// TIA Portal project "GirelloFB" (V16)

(* hardware
DEVICE "S7-1200 station_1"  S7-1200 Station
   slot 0: "Telaio di montaggio_0"  S7-1200 Rack  Rack  V1.0
   slot 1: "PLC_1"  CPU 1214C DC/DC/Rly  6ES7 214-1HG40-0XB0  V4.1
*)

// ===== PLC "PLC_1"  CPU 1214C DC/DC/Rly =====

VAR_GLOBAL   // PLC tag table "Tabella delle variabili standard"
   "START_1" AT %I0.0 : Bool;
   "S1_1" AT %I0.1 : Bool;
   "S2_1" AT %I0.2 : Bool;
   "S3_1" AT %I0.3 : Bool;
   "M_left_1" AT %Q0.0 : Bool;
   "M_right_1" AT %Q0.1 : Bool;
   "START_2" AT %I0.4 : Bool;
   "S1_2" AT %I0.5 : Bool;
   "S2_2" AT %I0.6 : Bool;
   "M_left_2" AT %Q0.2 : Bool;
   "M_right_2" AT %Q0.3 : Bool;
   "S3_2" AT %I0.7 : Bool;
END_VAR

VAR_GLOBAL CONSTANT   // PLC tag table "Tabella delle variabili standard"
   "TEMPO_TRASCORSO_T1_Girello1" : Time := T#3s;
   "TEMPO_TRASCORSO_T2_Girello1" : Time := T#8s;
   "TEMPO_TRASCORSO_T1_Girello2" : Time := T#5s;
   "TEMPO_TRASCORSO_T2_Girello2" : Time := T#10s;
END_VAR

DATA_BLOCK "Girello_DB_1"   // DB1
{ S7_Optimized_Access := 'TRUE' }
VERSION : 0.1
// stored: InstanceOfName Girello
"Girello"
BEGIN
END_DATA_BLOCK

DATA_BLOCK "Girello_DB_2"   // DB2
{ S7_Optimized_Access := 'TRUE' }
VERSION : 0.1
// stored: InstanceOfName Girello
"Girello"
BEGIN
END_DATA_BLOCK

FUNCTION_BLOCK "Girello"   // FB1, LAD
{ S7_Optimized_Access := 'TRUE' }
VERSION : 0.1
   VAR_INPUT
      START : Bool;
      S1 : Bool;
      S2 : Bool;
      S3 : Bool;
      TEMPO_TRASCORSO_T1 : Time;
      TEMPO_TRASCORSO_T2 : Time;
   END_VAR
   VAR_OUTPUT
      M_left : Bool;
      M_right : Bool;
   END_VAR
   VAR RETAIN
      HOME : Bool := true;
      ROTATE_TO_LEFT : Bool;
      POSITION_S2 : Bool;
      POSITION_S3 : Bool;
      ROTATE_TO_RIGHT : Bool;
   END_VAR
   VAR
      IEC_Timer_0_Instance_1 : TON_TIME;
      IEC_Timer_0_Instance_2 : TON_TIME;
   END_VAR
BEGIN

REGION Network 1
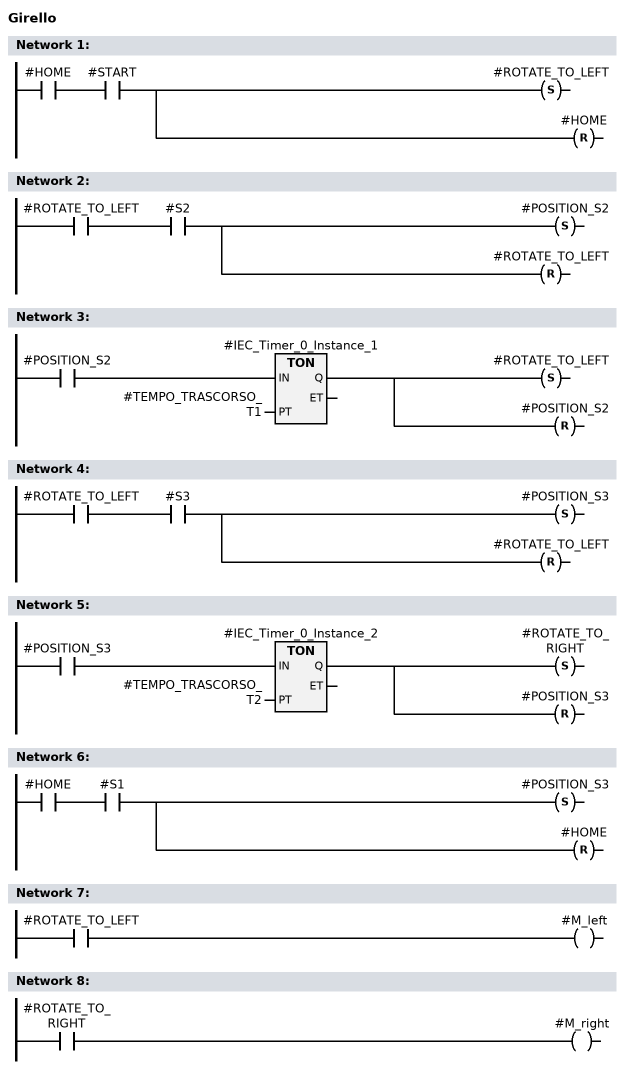
   RUNG wire#powerrail
      Contact( #HOME )
      Contact( #START )
      wire#w1
      S_Coil( #ROTATE_TO_LEFT )
   END_RUNG
   RUNG wire#w1
      R_Coil( #HOME )
   END_RUNG
   // the same network as SCL:
   IF #HOME AND #START THEN
       #ROTATE_TO_LEFT := TRUE;
       #HOME := FALSE;
   END_IF;
END_REGION

REGION Network 2
   RUNG wire#powerrail
      Contact( #ROTATE_TO_LEFT )
      Contact( #S2 )
      wire#w1
      S_Coil( #POSITION_S2 )
   END_RUNG
   RUNG wire#w1
      R_Coil( #ROTATE_TO_LEFT )
   END_RUNG
   // the same network as SCL:
   IF #ROTATE_TO_LEFT AND #S2 THEN
       #POSITION_S2 := TRUE;
       #ROTATE_TO_LEFT := FALSE;
   END_IF;
END_REGION

REGION Network 3
   #IEC_Timer_0_Instance_1(IN := #POSITION_S2, PT := #TEMPO_TRASCORSO_T1);   // TON
   IF #IEC_Timer_0_Instance_1.Q THEN
       #ROTATE_TO_LEFT := TRUE;
       #POSITION_S2 := FALSE;
   END_IF;
END_REGION

REGION Network 4
   RUNG wire#powerrail
      Contact( #ROTATE_TO_LEFT )
      Contact( #S3 )
      wire#w1
      S_Coil( #POSITION_S3 )
   END_RUNG
   RUNG wire#w1
      R_Coil( #ROTATE_TO_LEFT )
   END_RUNG
   // the same network as SCL:
   IF #ROTATE_TO_LEFT AND #S3 THEN
       #POSITION_S3 := TRUE;
       #ROTATE_TO_LEFT := FALSE;
   END_IF;
END_REGION

REGION Network 5
   #IEC_Timer_0_Instance_2(IN := #POSITION_S3, PT := #TEMPO_TRASCORSO_T2);   // TON
   IF #IEC_Timer_0_Instance_2.Q THEN
       #ROTATE_TO_RIGHT := TRUE;
       #POSITION_S3 := FALSE;
   END_IF;
END_REGION

REGION Network 6
   RUNG wire#powerrail
      Contact( #HOME )
      Contact( #S1 )
      wire#w1
      S_Coil( #POSITION_S3 )
   END_RUNG
   RUNG wire#w1
      R_Coil( #HOME )
   END_RUNG
   // the same network as SCL:
   IF #HOME AND #S1 THEN
       #POSITION_S3 := TRUE;
       #HOME := FALSE;
   END_IF;
END_REGION

REGION Network 7
   RUNG wire#powerrail
      Contact( #ROTATE_TO_LEFT )
      Coil( #M_left )
   END_RUNG
   // the same network as SCL:
   #M_left := #ROTATE_TO_LEFT;
END_REGION

REGION Network 8
   RUNG wire#powerrail
      Contact( #ROTATE_TO_RIGHT )
      Coil( #M_right )
   END_RUNG
   // the same network as SCL:
   #M_right := #ROTATE_TO_RIGHT;
END_REGION
END_FUNCTION_BLOCK

ORGANIZATION_BLOCK "Main"   // OB1, LAD, ProgramCycle
TITLE = "Main Program Sweep (Cycle)"
{ S7_Optimized_Access := 'TRUE' }
VERSION : 0.1
   VAR_INPUT
      Initial_Call : Bool;   // Initial call of this OB
      Remanence : Bool;   // =True, if remanent data are available
   END_VAR
BEGIN
END_ORGANIZATION_BLOCK

ORGANIZATION_BLOCK "Cyclic_Interrupt_50ms"   // OB30, LAD, CyclicInterrupt
{ S7_Optimized_Access := 'TRUE' }
VERSION : 0.1
   VAR_INPUT
      Initial_Call : Bool;   // Initial call of this OB
      Event_Count : Int;   // Events discarded
   END_VAR
BEGIN

REGION Network 1
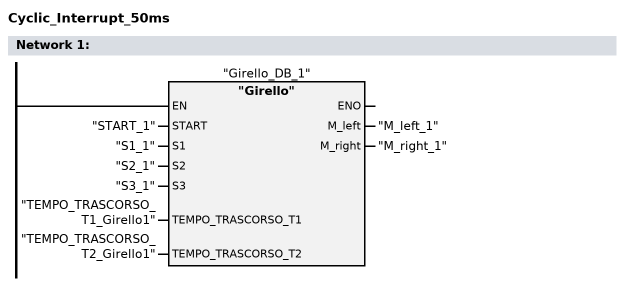
   RUNG wire#powerrail
      "Girello_DB_1"(START := "START_1", S1 := "S1_1", S2 := "S2_1", S3 := "S3_1", TEMPO_TRASCORSO_T1 := "TEMPO_TRASCORSO_T1_Girello1", TEMPO_TRASCORSO_T2 := "TEMPO_TRASCORSO_T2_Girello1", M_left => "M_left_1", M_right => "M_right_1")
   END_RUNG
   // the same network as SCL:
   "Girello_DB_1"(START := "START_1",   // "Girello"
                  S1 := "S1_1",
                  S2 := "S2_1",
                  S3 := "S3_1",
                  TEMPO_TRASCORSO_T1 := "TEMPO_TRASCORSO_T1_Girello1",
                  TEMPO_TRASCORSO_T2 := "TEMPO_TRASCORSO_T2_Girello1",
                  M_left => "M_left_1",
                  M_right => "M_right_1");
END_REGION
END_ORGANIZATION_BLOCK

ORGANIZATION_BLOCK "Cyclic_Interrupt_100ms"   // OB31, LAD, CyclicInterrupt
{ S7_Optimized_Access := 'TRUE' }
VERSION : 0.1
   VAR_INPUT
      Initial_Call : Bool;   // Initial call of this OB
      Event_Count : Int;   // Events discarded
   END_VAR
BEGIN

REGION Network 1
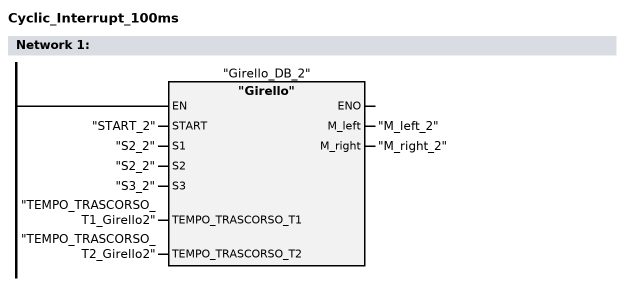
   RUNG wire#powerrail
      "Girello_DB_2"(START := "START_2", S1 := "S2_2", S2 := "S2_2", S3 := "S3_2", TEMPO_TRASCORSO_T1 := "TEMPO_TRASCORSO_T1_Girello2", TEMPO_TRASCORSO_T2 := "TEMPO_TRASCORSO_T2_Girello2", M_left => "M_left_2", M_right => "M_right_2")
   END_RUNG
   // the same network as SCL:
   "Girello_DB_2"(START := "START_2",   // "Girello"
                  S1 := "S2_2",
                  S2 := "S2_2",
                  S3 := "S3_2",
                  TEMPO_TRASCORSO_T1 := "TEMPO_TRASCORSO_T1_Girello2",
                  TEMPO_TRASCORSO_T2 := "TEMPO_TRASCORSO_T2_Girello2",
                  M_left => "M_left_2",
                  M_right => "M_right_2");
END_REGION
END_ORGANIZATION_BLOCK